FUNCTION_BLOCK MainStation EXTENDS TcoCore.TcoObject
//VAR
//    turckRfidHead : RfidHead(THIS^, T#1MS);
//    sUId          : T_MaxString;
//END_VAR
//VAR
//	    _uid          : BOOL;
//END_VAR

VAR
    //    rfidHead_Test : IVController_Test;

END_VAR

//TcUnit.RUN();

END_FUNCTION_BLOCK

(* stored: Version 1.1.0.1, ProductVersion 3.1.4024.12
   POU MainStation: Id {83331414-2fae-0cd4-0428-a092703db629}, SpecialFunc None *)
